FUNCTION_BLOCK MathFunc

METHOD Factorial : LREAL
VAR_INPUT
    n : INT;
END_VAR

VAR
	i : INT;
    result: INT := 1;
    
END_VAR
FOR i := 1 TO n DO
    result := result * i;
END_FOR

Factorial := result;
END_METHOD

METHOD FindForSixPoints : BOOL

VAR_INPUT
	start_pos : ARRAY [1..6] OF LREAL;
	final_pos : ARRAY [1..6] OF LREAL;
END_VAR

VAR_OUTPUT
	six_pos : ARRAY [1..6, 1..6] OF LREAL;
END_VAR

VAR
	i, j : DINT;
	delta : ARRAY[1..6] OF LREAL;
	section : ARRAY[1..5] OF LREAL;
	weight : ARRAY[1..5] OF LREAL := [15, 21, 25.5, 25, 13.5];
END_VAR
FOR i := 1 TO 6 DO
	delta[i] := final_pos[i] - start_pos[i];
	FOR j := 1 TO 5 DO
		section[j] := delta[i] * weight[j] / 100;
	END_FOR
	six_pos[1, i] := start_pos[i];
	FOR j := 2 TO 6 DO
		six_pos[j, i] := six_pos[j - 1, i] + section[j - 1];
	END_FOR		
END_FOR
END_METHOD

METHOD FindFullTime : BOOL

VAR_INPUT
	pos01 : ARRAY [1..3] OF LREAL;
	pos02 : ARRAY [1..3] OF LREAL;
	time_factor : LREAL;
END_VAR

VAR_OUTPUT
	execute_fullTime : LREAL;
END_VAR

VAR
	longest_distance : LREAL;
END_VAR
longest_distance := SQRT(EXPT(pos02[1] - pos01[1], 2) + EXPT(pos02[2] - pos01[2], 2) + EXPT(pos02[3] - pos01[3], 2)); 
execute_fullTime := EXPT(time_factor, -1) * longest_distance;

//fix time proble
execute_fullTime := LREAL_TO_DINT(execute_fullTime * EXPT(10, 7))/EXPT(10, 7);
END_METHOD

METHOD GaussianElimination

// n-order trajectory curve fitting
VAR_IN_OUT
	base_mat : ARRAY[*, *] OF LREAL;    // 6 of time-related function(Assume t0 at last row)
	extend_mat : ARRAY[*, *] OF LREAL;  // target(XYZRPY) on corresponding time
	temp_mat : ARRAY[*, *] OF LREAL;  	// 暫存矩陣(放單位矩陣跟反矩陣)
END_VAR

VAR_INPUT
	order : INT;
END_VAR

VAR
	n : INT;
	row : INT;
	column : INT;
	gain : LREAL;
	temp : LREAL;
	base_mat_Copy : ARRAY [1..6] OF ARRAY [1..6] OF LREAL;
END_VAR
FOR row := 1 TO order DO
	FOR column := 1 TO order DO
		base_mat_Copy[row][column] := base_mat[row, column];
	END_FOR
END_FOR
// Create a unit
FOR row := 1 TO order DO
	FOR column := 1 TO order DO
		IF row = column THEN
			temp_mat[row, column] := 1;
		ELSE
			temp_mat[row, column] := 0;
		END_IF
	END_FOR
END_FOR

// Lower triangle to zeros
FOR n := 1 TO order DO
	FOR row := n+1 TO order DO
		gain := base_mat[row, n] / base_mat[n, n];
		// Elimination
		FOR column := 1 TO order DO
			base_mat[row, column] := base_mat[row, column] - gain * base_mat[n, column];
			// The matrix shape is exacly the same as base_mat
			temp_mat[row, column] := temp_mat[row, column] - gain * temp_mat[n, column];
		END_FOR
	END_FOR
END_FOR

// Upper triangle to zeros
FOR n := order TO 1 BY -1 DO
	FOR row := n-1 TO 1 BY -1 DO
		gain := base_mat[row, n] / base_mat[n, n];
		// Elimination
		FOR column := order TO 1 BY -1 DO
			base_mat[row, column] := base_mat[row, column] - gain * base_mat[n, column];
			// The matrix shape is exacly the same as base_mat
			temp_mat[row, column] := temp_mat[row, column] - gain * temp_mat[n, column];
		END_FOR
	END_FOR
END_FOR

// Solve equation
FOR row := 1 TO 6 DO
	FOR column := 1 TO 6 DO
		temp_mat[row, column] := temp_mat[row, column] / base_mat[row, row];
		//Round(num1 := temp_mat[row, column], n := 2, num2 => temp_mat[row, column]);
	END_FOR
END_FOR
MultiplyByMatrix(A := extend_mat, B := temp_mat, C := base_mat, n := 6);

// Switch the name of matrix
FOR row := 1 TO order DO
	FOR column := 1 TO order DO
		temp := temp_mat[row, column];
		temp_mat[row, column] := base_mat[row, column];
		base_mat[row, column] := temp;
	END_FOR		
END_FOR
END_METHOD

METHOD MultiplyByMatrix : BOOL

VAR_IN_OUT
	A : ARRAY[*, *] OF LREAL;
	B : ARRAY[*, *] OF LREAL;
	C : ARRAY[*, *] OF LREAL;
END_VAR

VAR_INPUT
	n : INT;
END_VAR

VAR 
	i: DINT;   // row
	j : DINT;  // col
	k : Dint;  // order
END_VAR
FOR i := 1 TO n DO
	FOR j := 1 TO n DO
		C[i, j] := 0;
	END_FOR
END_FOR

FOR i := 1 TO n DO
	FOR j := 1 TO n DO
		FOR k := 1 TO n DO
			C[i, j] := C[i, j] + A[i, k] * B[k, j];
			//Round(num1 := C[i, j], n := 5, num2 => C[i, j]);
		END_FOR
	END_FOR
END_FOR
END_METHOD

METHOD Round : BOOL
VAR_INPUT
	num1 : LREAL;
	n : INT;
END_VAR

VAR_OUTPUT
	num2 : lreal;
END_VAR
num2 := LREAL_TO_DINT(num1 * EXPT(10, n) ) / EXPT(10, n);
END_METHOD

METHOD VectorMotionPOS : BOOL

VAR_IN_OUT
	POS : ARRAY [AXIS_MIN_IDX..AXIS_MAX_IDX] OF LREAL;
END_VAR

VAR_INPUT
	Direcation : LREAL;
	Path_Motion_Displace : LREAL;
END_VAR
IF Direcation = 1 THEN
	POS[1] := POS[1] + Path_Motion_Displace;
ELSIF Direcation = 2 THEN
	POS[2] := POS[2] + Path_Motion_Displace;
ELSIF Direcation = 3 THEN
	POS[3] := POS[3] + Path_Motion_Displace;
ELSIF Direcation = 4 THEN
	POS[1] := POS[1] + Path_Motion_Displace * 0.5 * EXPT(2, 0.5);
	POS[2] := POS[2] + Path_Motion_Displace * 0.5 * EXPT(2, 0.5);
ELSIF Direcation = 5 THEN
	POS[1] := POS[1] + Path_Motion_Displace * 0.5 * EXPT(2, 0.5);
	POS[2] := POS[2] - Path_Motion_Displace * 0.5 * EXPT(2, 0.5);
END_IF
END_METHOD

END_FUNCTION_BLOCK

(* stored: Version 1.1.0.1, ProductVersion 3.1.4024.13
   POU MathFunc: Id {0948e163-60a5-441c-8e57-745d9d01a6b2}, SpecialFunc None
   Method Factorial: Id {6e134467-a6b1-430b-9b8c-6f4b66abd488}
   Method FindForSixPoints: Id {f6602cd8-15c6-4c12-bdf1-c87fd0b2d5c7}
   Method FindFullTime: Id {73e052dc-8b2b-46af-9c41-5d3805da2579}
   Method GaussianElimination: Id {d17d2efb-cab2-4248-ab5f-053d253678d2}
   Method MultiplyByMatrix: Id {d43ac27a-3014-4b06-9cee-ce786a9c0bbb}
   Method Round: Id {f0f879cb-633b-4858-a892-d1ba22afd6ed}
   Method VectorMotionPOS: Id {4be0ed86-e5fb-44ae-ad62-944db606b416} *)
